(* Schneider Machine Expert - Basic project Master AHU Mod TCP, file version 2.2.0.0 *)
(* ProjectInformations: Name=New project *)

HARDWARE
  Cpu 0: TM221ME16R/G
  ModuleExtensionObject 0: TM3AI8/G
  EthernetConfiguration: NetworkName=M221, IpAllocationMode=FixedAddress, IpAddress=10.3.12.250, SubnetMask=255.255.252.0
  SerialLineConfiguration: Baud=Baud9600, Parity=ParityEven, DataBits=DataBits8, StopBits=StopBits1, PhysicalMedium=PhysicalMediumRs485, TransmissionMode=TransmissionModeModbusRtu, SlaveId=1, Addressing=MasterAddressing
  MastTask: UsePeriodScanMode=false, PeriodScan=100
  FastTask: Period=255
  CpuBehavior: StartingMode=StartAsPreviousState, AutoSaveRamOnEeprom=true, WatchdogPeriod=250

SYMBOLS  (address, symbol, comment, settings)
  %M14      ERR_SLAVE_1
  %M15      ERR_SLAVE_2
  %M20      ERR_SERIAL_1
  %M21      ERR_SERIAL_2
  %M22      ERR_SERIAL_3
  %M23      ERR_SERIAL_4
  %M24      ERR_SERIAL_5
  %M25      ERR_SERIAL_6
  %M26      ERR_SERIAL_7
  %M27      ERR_SERIAL_8
  %S12      SB_RUNMODE  "The controller is running"
  %MW0      SENSOR_TEMP_0910
  %MW1      SENSOR_TEMP_1112
  %MW2      SENSOR_HUMI_0910
  %MW3      SENSOR_HUMI_1112
  %MW5      SENSOR_TEMP_1314
  %MW6      SENSOR_TEMP_1516
  %MW7      SENSOR_HUMI_1314
  %MW8      SENSOR_HUMI_1516
  %TM0        [Preset=3, Base=OneSecond]
  %TM1        [Preset=3, Base=OneSecond]
  %TM2        [Preset=5, Base=OneHundredMilliSeconds]
  %TM4        [Type=TOF, Preset=10, Base=OneHundredMilliSeconds]
  %READ_VAR0   [Link(Value(FBComLinkParameterEnums=SerialLine1)), RemoteDeviceId(Value(int=9)), Timeout(Value(int=100)), ObjType(Value(FBComObjTypeParameterEnums=IW)), FirstObj(Value(int=0)), Quantity(Value(int=1)), IndexData(Value(int=20))]
  %READ_VAR1   [Link(Value(FBComLinkParameterEnums=SerialLine1)), RemoteDeviceId(Value(int=10)), Timeout(Value(int=100)), ObjType(Value(FBComObjTypeParameterEnums=IW)), FirstObj(Value(int=0)), Quantity(Value(int=1)), IndexData(Value(int=21))]
  %READ_VAR2   [Link(Value(FBComLinkParameterEnums=SerialLine1)), RemoteDeviceId(Value(int=11)), Timeout(Value(int=100)), ObjType(Value(FBComObjTypeParameterEnums=IW)), FirstObj(Value(int=0)), Quantity(Value(int=1)), IndexData(Value(int=22))]
  %READ_VAR3   [Link(Value(FBComLinkParameterEnums=SerialLine1)), RemoteDeviceId(Value(int=12)), Timeout(Value(int=100)), ObjType(Value(FBComObjTypeParameterEnums=IW)), FirstObj(Value(int=0)), Quantity(Value(int=1)), IndexData(Value(int=23))]
  %READ_VAR4   [Link(Value(FBComLinkParameterEnums=SerialLine1)), RemoteDeviceId(Value(int=13)), Timeout(Value(int=200)), ObjType(Value(FBComObjTypeParameterEnums=IW)), FirstObj(Value(int=0)), Quantity(Value(int=1)), IndexData(Value(int=24))]
  %READ_VAR5   [Link(Value(FBComLinkParameterEnums=SerialLine1)), RemoteDeviceId(Value(int=14)), Timeout(Value(int=100)), ObjType(Value(FBComObjTypeParameterEnums=IW)), FirstObj(Value(int=0)), Quantity(Value(int=1)), IndexData(Value(int=25))]
  %READ_VAR6   [Link(Value(FBComLinkParameterEnums=SerialLine1)), RemoteDeviceId(Value(int=15)), Timeout(Value(int=200)), ObjType(Value(FBComObjTypeParameterEnums=IW)), FirstObj(Value(int=0)), Quantity(Value(int=1)), IndexData(Value(int=26))]
  %READ_VAR7   [Link(Value(FBComLinkParameterEnums=SerialLine1)), RemoteDeviceId(Value(int=16)), Timeout(Value(int=100)), ObjType(Value(FBComObjTypeParameterEnums=IW)), FirstObj(Value(int=0)), Quantity(Value(int=1)), IndexData(Value(int=27))]
  %Q0.0     STATUS_
  %IW1.0    TEMP_LINE_09_10  "Sensor Temperature Line 09-10 (Lantai 1)"  [Type=Type_4_20mA, Scope=Scope_Customized, Minimum=4000, Maximum=20000]
  %IW1.1    HUM_LINE_09_10  "Sensor Humidity Line 09-10 (Lantai 1)"  [Type=Type_4_20mA, Scope=Scope_Customized, Minimum=4000, Maximum=20000]
  %IW1.2    TEMP_LINE_11_12  "Sensor Temperature Line 11-12 (Lantai 1)"  [Type=Type_4_20mA, Scope=Scope_Customized, Minimum=4000, Maximum=20000]
  %IW1.3    HUM_LINE_11_12  "Sensor Humidity  Line 11-12 (Lantai 1)"  [Type=Type_4_20mA, Scope=Scope_Customized, Minimum=4000, Maximum=20000]
  %IW1.4    TEMP_LINE_13_14  "Sensor Temperature Line 13-14 (Lantai 1)"  [Type=Type_4_20mA, Scope=Scope_Customized, Minimum=4000, Maximum=20000]
  %IW1.5    HUM_LINE_13_14  "Sensor Humidity Line 13-14 (Lantai 1)"  [Type=Type_4_20mA, Scope=Scope_Customized, Minimum=4000, Maximum=20000]
  %IW1.6    TEMP_LINE_15_16  "Sensor Temperature Line 15-16 (Lantai 1)"  [Type=Type_4_20mA, Scope=Scope_Customized, Minimum=4000, Maximum=20000]
  %IW1.7    HUM_LINE_15_16  "Sensor Humidity Line 15-16 (Lantai 1)"  [Type=Type_4_20mA, Scope=Scope_Customized, Minimum=4000, Maximum=20000]

POU CONTROL  SERIAL
  (* SectionNumber=1 *)

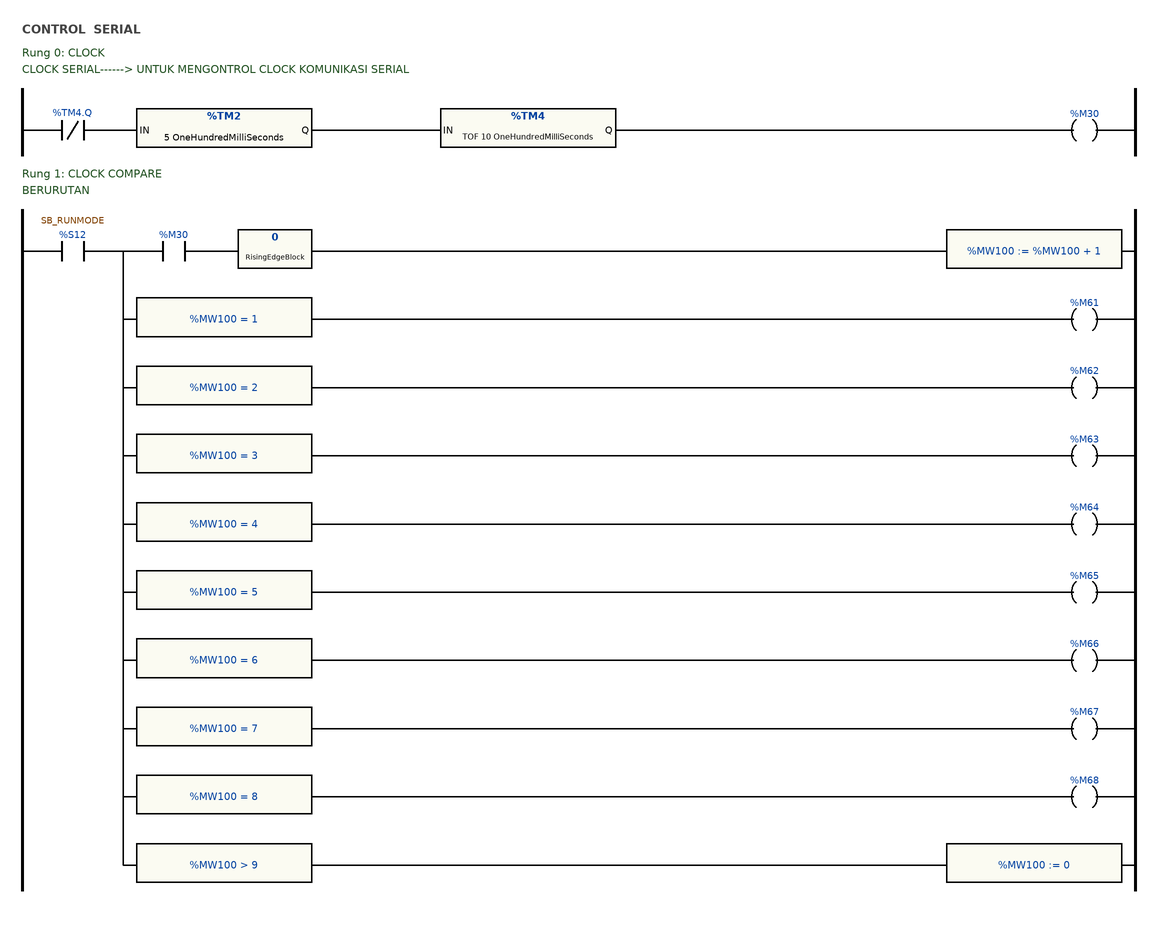

// Rung 0: CLOCK
// CLOCK SERIAL------> UNTUK MENGONTROL CLOCK KOMUNIKASI SERIAL
  LD 1
  MULTIFB
  BLK %TM2
  LDN %TM4.Q
  IN
  OUT_BLK
  LD Q
  ST %MW2000:X0
  END_BLK
  BLK %TM4
  LD %MW2000:X0
  IN
  OUT_BLK
  LD Q
  ST %M30
  END_BLK
  MULTIFB
  // as ST:
  //   %TM2(IN := NOT %TM4.Q);
  //   %TM4(IN := %TM2.Q);
  //   %M30 := %TM4.Q;

// Rung 1: CLOCK COMPARE
// BERURUTAN
  LD %S12                 (* SB_RUNMODE *)
  MPS
  AND %M30
  RISING0
  [ %MW100 := %MW100 + 1 ]
  MRD
  AND [ %MW100 = 1 ]
  ST %M61
  MRD
  AND [ %MW100 = 2 ]
  ST %M62
  MRD
  AND [ %MW100 = 3 ]
  ST %M63
  MRD
  AND [ %MW100 = 4 ]
  ST %M64
  MRD
  AND [ %MW100 = 5 ]
  ST %M65
  MRD
  AND [ %MW100 = 6 ]
  ST %M66
  MRD
  AND [ %MW100 = 7 ]
  ST %M67
  MRD
  AND [ %MW100 = 8 ]
  ST %M68
  MPP
  AND [ %MW100 > 9 ]
  [ %MW100 := 0 ]
  // as ST:
  //   IF RISING(SB_RUNMODE AND %M30) THEN %MW100 := %MW100 + 1; END_IF;
  //   %M61 := SB_RUNMODE AND %MW100 = 1;
  //   %M62 := SB_RUNMODE AND %MW100 = 2;
  //   %M63 := SB_RUNMODE AND %MW100 = 3;
  //   %M64 := SB_RUNMODE AND %MW100 = 4;
  //   %M65 := SB_RUNMODE AND %MW100 = 5;
  //   %M66 := SB_RUNMODE AND %MW100 = 6;
  //   %M67 := SB_RUNMODE AND %MW100 = 7;
  //   %M68 := SB_RUNMODE AND %MW100 = 8;
  //   IF SB_RUNMODE AND %MW100 > 9 THEN %MW100 := 0; END_IF;

POU READ  SERIAL
  (* SectionNumber=2 *)

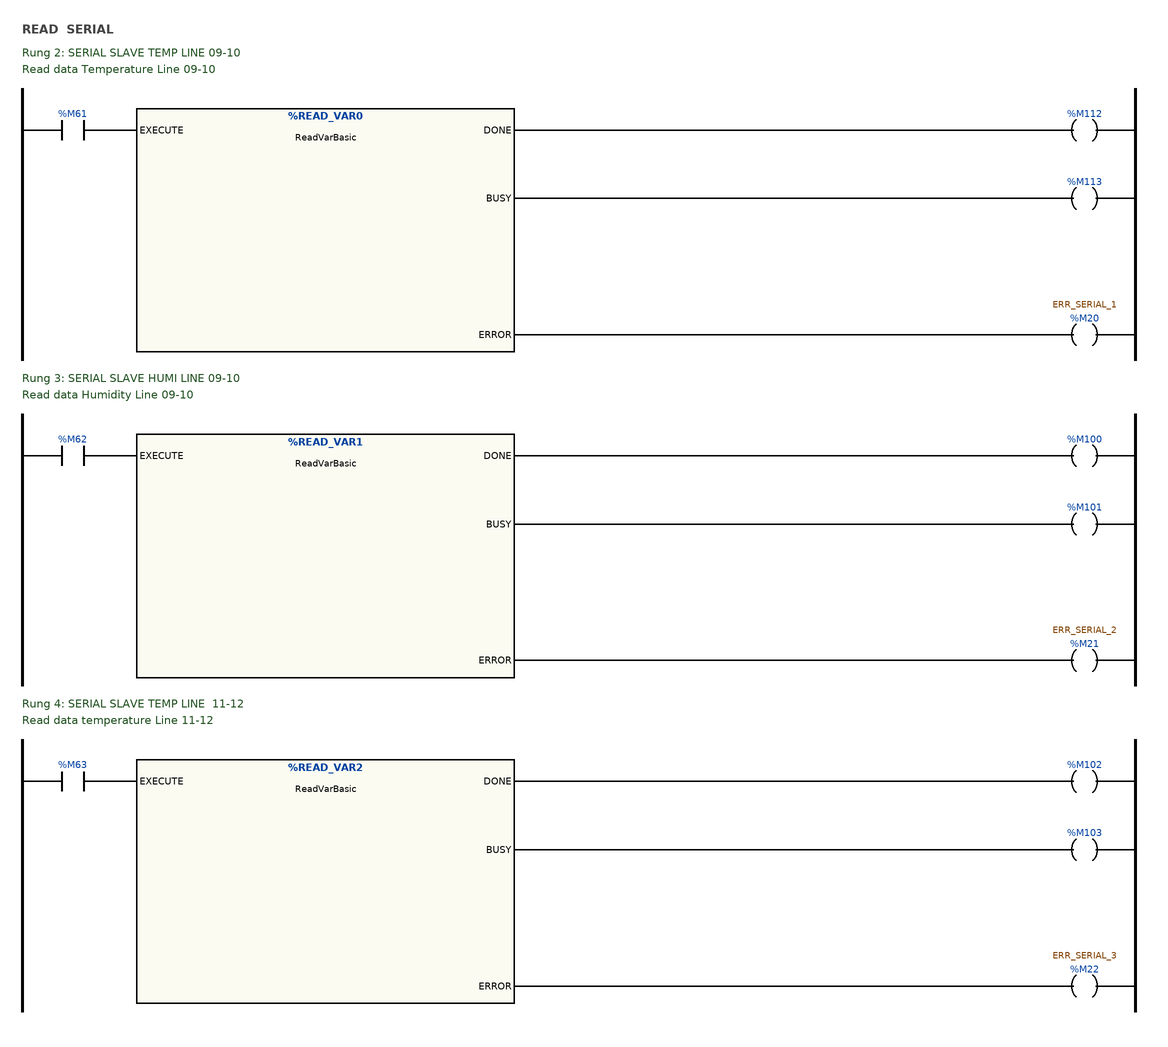

// Rung 2: SERIAL SLAVE TEMP LINE 09-10
// Read data Temperature Line 09-10
  BLK %READ_VAR0
  LD %M61
  EXECUTE
  OUT_BLK
  LD DONE
  ST %M112
  LD BUSY
  ST %M113
  LD ERROR
  ST %M20                 (* ERR_SERIAL_1 *)
  END_BLK
  // as ST:
  //   %READ_VAR0(EXECUTE := %M61);
  //   %M112 := %READ_VAR0.DONE;
  //   %M113 := %READ_VAR0.BUSY;
  //   ERR_SERIAL_1 := %READ_VAR0.ERROR;

// Rung 3: SERIAL SLAVE HUMI LINE 09-10
// Read data Humidity Line 09-10
  BLK %READ_VAR1
  LD %M62
  EXECUTE
  OUT_BLK
  LD DONE
  ST %M100
  LD BUSY
  ST %M101
  LD ERROR
  ST %M21                 (* ERR_SERIAL_2 *)
  END_BLK
  // as ST:
  //   %READ_VAR1(EXECUTE := %M62);
  //   %M100 := %READ_VAR1.DONE;
  //   %M101 := %READ_VAR1.BUSY;
  //   ERR_SERIAL_2 := %READ_VAR1.ERROR;

// Rung 4: SERIAL SLAVE TEMP LINE  11-12
// Read data temperature Line 11-12
  BLK %READ_VAR2
  LD %M63
  EXECUTE
  OUT_BLK
  LD DONE
  ST %M102
  LD BUSY
  ST %M103
  LD ERROR
  ST %M22                 (* ERR_SERIAL_3 *)
  END_BLK
  // as ST:
  //   %READ_VAR2(EXECUTE := %M63);
  //   %M102 := %READ_VAR2.DONE;
  //   %M103 := %READ_VAR2.BUSY;
  //   ERR_SERIAL_3 := %READ_VAR2.ERROR;

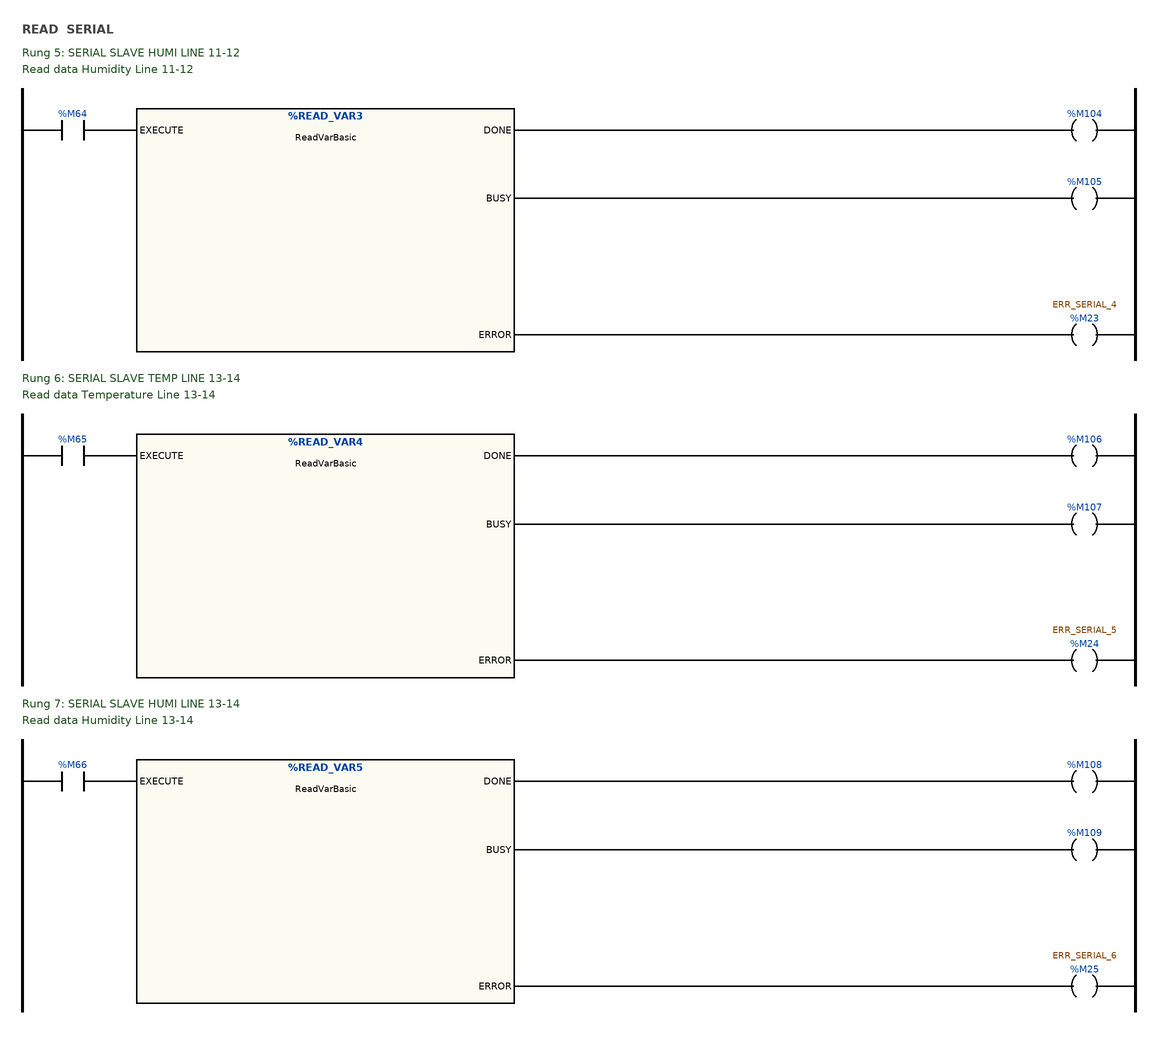

// Rung 5: SERIAL SLAVE HUMI LINE 11-12
// Read data Humidity Line 11-12
  BLK %READ_VAR3
  LD %M64
  EXECUTE
  OUT_BLK
  LD DONE
  ST %M104
  LD BUSY
  ST %M105
  LD ERROR
  ST %M23                 (* ERR_SERIAL_4 *)
  END_BLK
  // as ST:
  //   %READ_VAR3(EXECUTE := %M64);
  //   %M104 := %READ_VAR3.DONE;
  //   %M105 := %READ_VAR3.BUSY;
  //   ERR_SERIAL_4 := %READ_VAR3.ERROR;

// Rung 6: SERIAL SLAVE TEMP LINE 13-14
// Read data Temperature Line 13-14
  BLK %READ_VAR4
  LD %M65
  EXECUTE
  OUT_BLK
  LD DONE
  ST %M106
  LD BUSY
  ST %M107
  LD ERROR
  ST %M24                 (* ERR_SERIAL_5 *)
  END_BLK
  // as ST:
  //   %READ_VAR4(EXECUTE := %M65);
  //   %M106 := %READ_VAR4.DONE;
  //   %M107 := %READ_VAR4.BUSY;
  //   ERR_SERIAL_5 := %READ_VAR4.ERROR;

// Rung 7: SERIAL SLAVE HUMI LINE 13-14
// Read data Humidity Line 13-14
  BLK %READ_VAR5
  LD %M66
  EXECUTE
  OUT_BLK
  LD DONE
  ST %M108
  LD BUSY
  ST %M109
  LD ERROR
  ST %M25                 (* ERR_SERIAL_6 *)
  END_BLK
  // as ST:
  //   %READ_VAR5(EXECUTE := %M66);
  //   %M108 := %READ_VAR5.DONE;
  //   %M109 := %READ_VAR5.BUSY;
  //   ERR_SERIAL_6 := %READ_VAR5.ERROR;

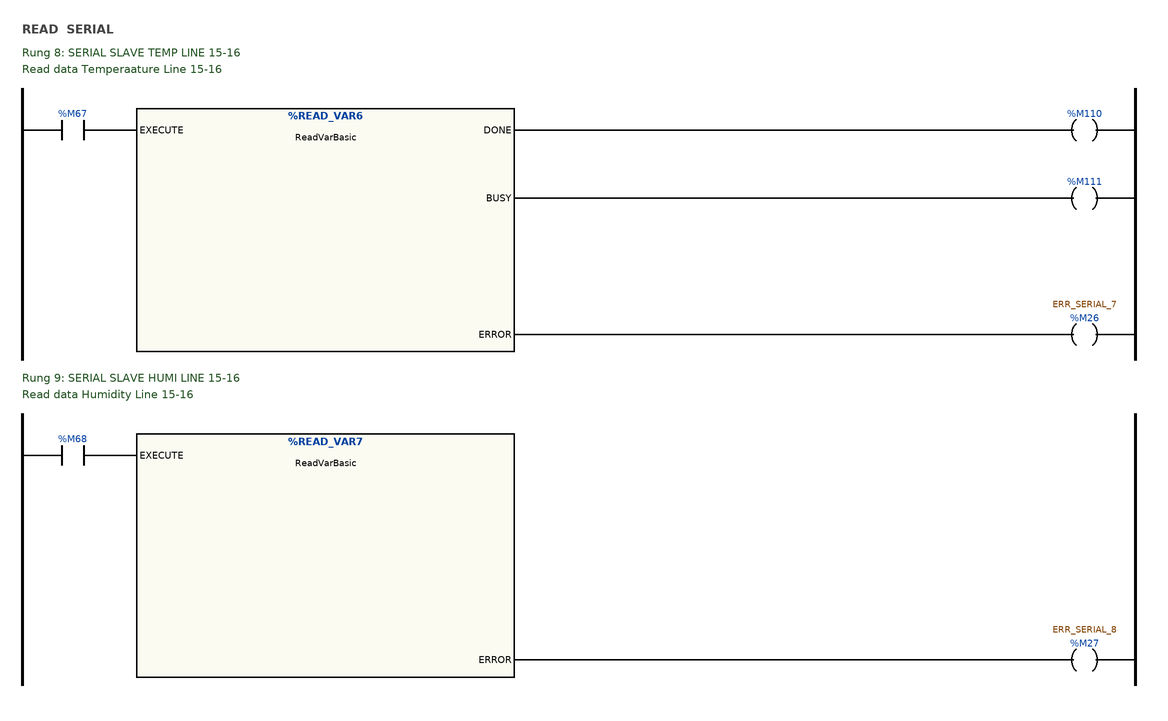

// Rung 8: SERIAL SLAVE TEMP LINE 15-16
// Read data Temperaature Line 15-16
  BLK %READ_VAR6
  LD %M67
  EXECUTE
  OUT_BLK
  LD DONE
  ST %M110
  LD BUSY
  ST %M111
  LD ERROR
  ST %M26                 (* ERR_SERIAL_7 *)
  END_BLK
  // as ST:
  //   %READ_VAR6(EXECUTE := %M67);
  //   %M110 := %READ_VAR6.DONE;
  //   %M111 := %READ_VAR6.BUSY;
  //   ERR_SERIAL_7 := %READ_VAR6.ERROR;

// Rung 9: SERIAL SLAVE HUMI LINE 15-16
// Read data Humidity Line 15-16
  BLK %READ_VAR7
  LD %M68
  EXECUTE
  OUT_BLK
  LD ERROR
  ST %M27                 (* ERR_SERIAL_8 *)
  END_BLK
  // as ST:
  //   %READ_VAR7(EXECUTE := %M68);
  //   ERR_SERIAL_8 := %READ_VAR7.ERROR;

POU MAIN PROGRAM MASTER AHU TCP
  (* SectionNumber=3 *)

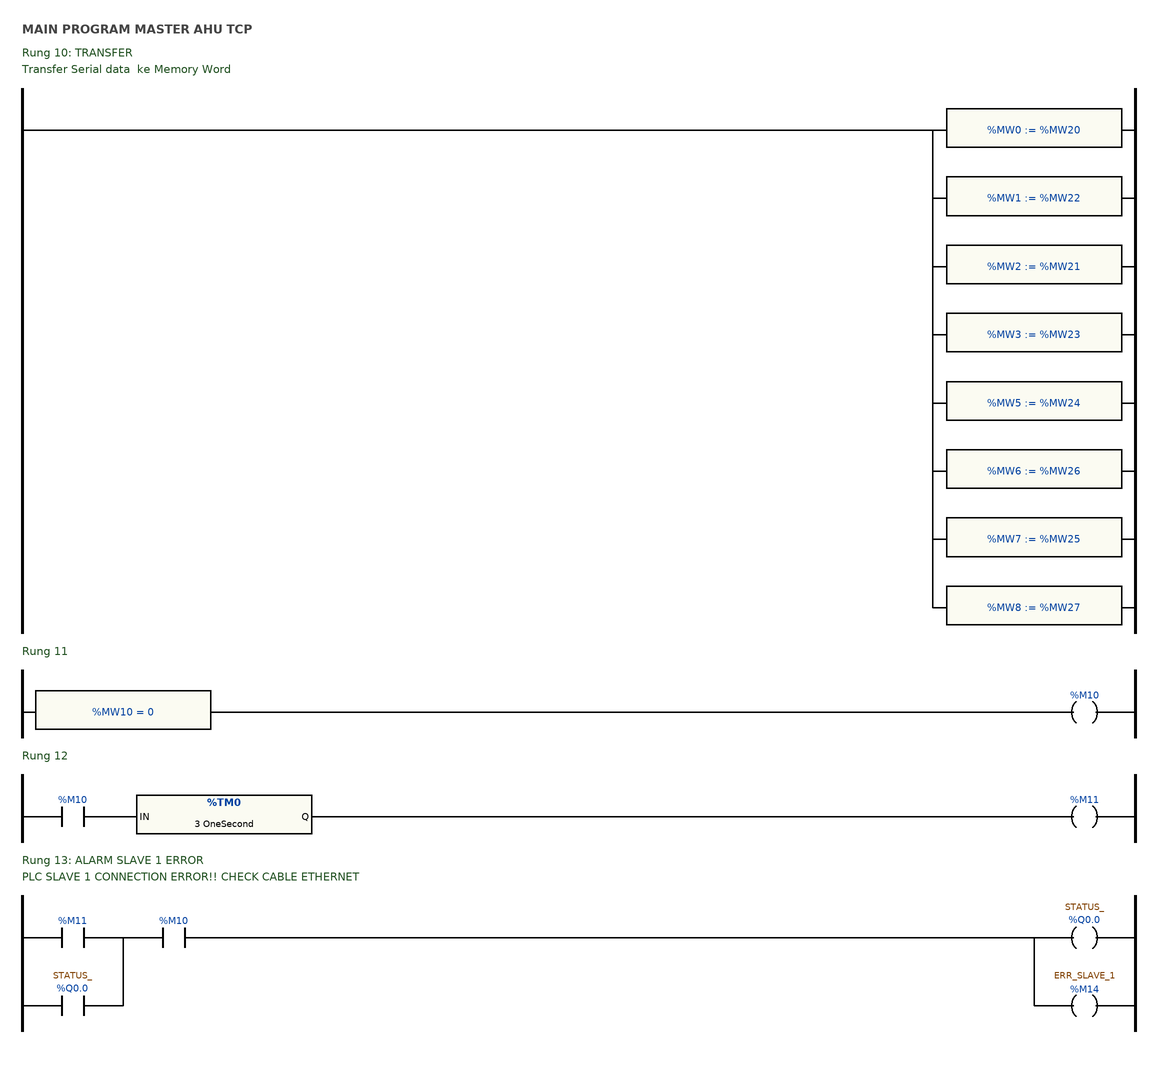

// Rung 10: TRANSFER
// Transfer Serial data  ke Memory Word
  LD 1
  [ %MW0 := %MW20 ]       (* SENSOR_TEMP_0910 *)
  [ %MW1 := %MW22 ]       (* SENSOR_TEMP_1112 *)
  [ %MW2 := %MW21 ]       (* SENSOR_HUMI_0910 *)
  [ %MW3 := %MW23 ]       (* SENSOR_HUMI_1112 *)
  [ %MW5 := %MW24 ]       (* SENSOR_TEMP_1314 *)
  [ %MW6 := %MW26 ]       (* SENSOR_TEMP_1516 *)
  [ %MW7 := %MW25 ]       (* SENSOR_HUMI_1314 *)
  [ %MW8 := %MW27 ]       (* SENSOR_HUMI_1516 *)
  // as ST:
  //   SENSOR_TEMP_0910 := %MW20;
  //   SENSOR_TEMP_1112 := %MW22;
  //   SENSOR_HUMI_0910 := %MW21;
  //   SENSOR_HUMI_1112 := %MW23;
  //   SENSOR_TEMP_1314 := %MW24;
  //   SENSOR_TEMP_1516 := %MW26;
  //   SENSOR_HUMI_1314 := %MW25;
  //   SENSOR_HUMI_1516 := %MW27;

// Rung 11
  LD [ %MW10 = 0 ]
  ST %M10
  // as ST:
  //   %M10 := %MW10 = 0;

// Rung 12
  BLK %TM0
  LD %M10
  IN
  OUT_BLK
  LD Q
  ST %M11
  END_BLK
  // as ST:
  //   %TM0(IN := %M10);
  //   %M11 := %TM0.Q;

// Rung 13: ALARM SLAVE 1 ERROR
// PLC SLAVE 1 CONNECTION ERROR!! CHECK CABLE ETHERNET
  LD %M11
  OR %Q0.0                (* STATUS_ *)
  AND %M10
  ST %Q0.0                (* STATUS_ *)
  ST %M14                 (* ERR_SLAVE_1 *)
  // as ST:
  //   _t1 := (%M11 OR STATUS_) AND %M10;
  //   STATUS_ := _t1;
  //   ERR_SLAVE_1 := _t1;

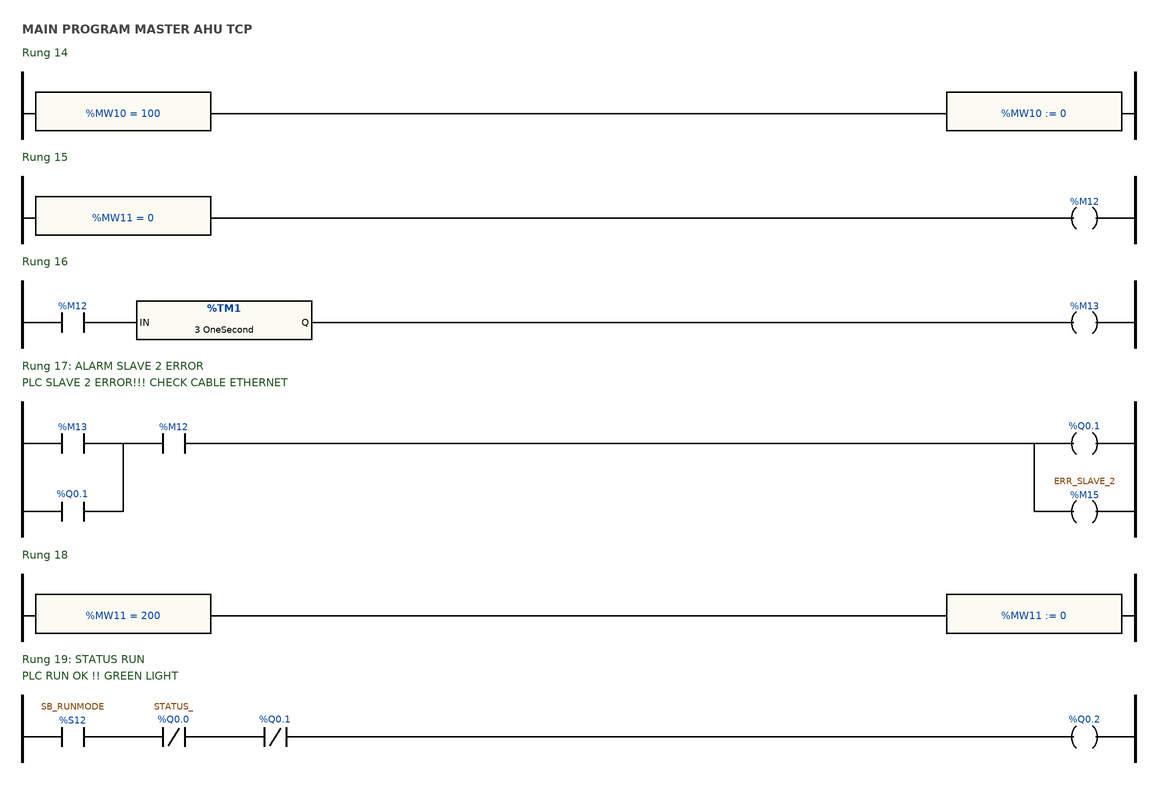

// Rung 14
  LD [ %MW10 = 100 ]
  [ %MW10 := 0 ]
  // as ST:
  //   IF %MW10 = 100 THEN %MW10 := 0; END_IF;

// Rung 15
  LD [ %MW11 = 0 ]
  ST %M12
  // as ST:
  //   %M12 := %MW11 = 0;

// Rung 16
  BLK %TM1
  LD %M12
  IN
  OUT_BLK
  LD Q
  ST %M13
  END_BLK
  // as ST:
  //   %TM1(IN := %M12);
  //   %M13 := %TM1.Q;

// Rung 17: ALARM SLAVE 2 ERROR
// PLC SLAVE 2 ERROR!!! CHECK CABLE ETHERNET
  LD %M13
  OR %Q0.1
  AND %M12
  ST %Q0.1
  ST %M15                 (* ERR_SLAVE_2 *)
  // as ST:
  //   _t1 := (%M13 OR %Q0.1) AND %M12;
  //   %Q0.1 := _t1;
  //   ERR_SLAVE_2 := _t1;

// Rung 18
  LD [ %MW11 = 200 ]
  [ %MW11 := 0 ]
  // as ST:
  //   IF %MW11 = 200 THEN %MW11 := 0; END_IF;

// Rung 19: STATUS RUN
// PLC RUN OK !! GREEN LIGHT
  LD %S12                 (* SB_RUNMODE *)
  ANDN %Q0.0              (* STATUS_ *)
  ANDN %Q0.1
  ST %Q0.2
  // as ST:
  //   %Q0.2 := SB_RUNMODE AND NOT STATUS_ AND NOT %Q0.1;
